// TIA Portal V19 export
TYPE "PII - BCM R15E-001-DI00-01,5-S4"
   STRUCT
      "Vibration Acceleration - Vibration Acceleration RMS a-RMS X" : Real;
      "Vibration Acceleration - Vibration Acceleration RMS a-RMS Y" : Real;
      "Vibration Acceleration - Vibration Acceleration RMS a-RMS Z" : Real;
      "Vibration Acceleration - Contact Temperature Contact Temperature" : Real;
      "Vibration Acceleration - Status Bits Main-Alarm a-RMS Magnitude Status" : Bool;
      "Vibration Acceleration - Status Bits Pre-Alarm a-RMS Magnitude Status" : Bool;
      "Vibration Acceleration - Status Bits Main-Alarm a-RMS Z Status" : Bool;
      "Vibration Acceleration - Status Bits Pre-Alarm a-RMS Z Status" : Bool;
      "Vibration Acceleration - Status Bits Main-Alarm a-RMS Y Status" : Bool;
      "Vibration Acceleration - Status Bits Pre-Alarm a-RMS Y Status" : Bool;
      "Vibration Acceleration - Status Bits Main-Alarm a-RMS X Status" : Bool;
      "Vibration Acceleration - Status Bits Pre-Alarm a-RMS X Status" : Bool;
      "Vibration Acceleration - Status Bits Main-Alarm v-RMS Magnitude Status" : Bool;
      "Vibration Acceleration - Status Bits Pre-Alarm v-RMS Magnitude Status" : Bool;
      "Vibration Acceleration - Status Bits Main-Alarm v-RMS Z Status" : Bool;
      "Vibration Acceleration - Status Bits Pre-Alarm v-RMS Z Status" : Bool;
      "Vibration Acceleration - Status Bits Main-Alarm v-RMS Y Status" : Bool;
      "Vibration Acceleration - Status Bits Pre-Alarm v-RMS Y Status" : Bool;
      "Vibration Acceleration - Status Bits Main-Alarm v-RMS X Status" : Bool;
      "Vibration Acceleration - Status Bits Pre-Alarm v-RMS X Status" : Bool;
      "Vibration Acceleration - Status Bits Reserved" : Bool;
      "Vibration Acceleration - Status Bits Reserved_1" : Bool;
      "Vibration Acceleration - Status Bits Reserved_2" : Bool;
      "Vibration Acceleration - Status Bits Vibration Severity Zone D" : Bool;
      "Vibration Acceleration - Status Bits Vibration Severity Zone C" : Bool;
      "Vibration Acceleration - Status Bits Vibration Severity Zone B" : Bool;
      "Vibration Acceleration - Status Bits Vibration Severity Zone A" : Bool;
      "Vibration Acceleration - Status Bits Reserved_3" : Bool;
      "Vibration Acceleration - Status Bits Reserved_4" : Bool;
      "Vibration Acceleration - Status Bits Reserved_5" : Bool;
      "Vibration Acceleration - Status Bits Reserved_6" : Bool;
      "Vibration Acceleration - Status Bits Reserved_7" : Bool;
      "Vibration Acceleration - Status Bits Reserved_8" : Bool;
      "Vibration Acceleration - Status Bits Reserved_9" : Bool;
      "Vibration Acceleration - Status Bits Contact Temperature Upper Alarm Status" : Bool;
      "Vibration Acceleration - Status Bits Contact Temperature Lower Alarm Status" : Bool;
      "Reserved Byte" : Bool;
      "Reserved Byte_1" : Bool;
      "Reserved Byte_2" : Bool;
      "Reserved Byte_3" : Bool;
      "Reserved Byte_4" : Bool;
      "Reserved Byte_5" : Bool;
      "Reserved Byte_6" : Bool;
      "Reserved Byte_7" : Bool;
      "Reserved Byte_8" : Bool;
      "Reserved Byte_9" : Bool;
      "Reserved Byte_10" : Bool;
      "Reserved Byte_11" : Bool;
      "Port qualifier" : Byte;
   END_STRUCT;
END_TYPE
